# EPICS autosave request: urRobotApp/Db/waypointL_settings.req
$(P)WaypointL:$(N).VAL
$(P)WaypointL:$(N):X.VAL
$(P)WaypointL:$(N):Y.VAL
$(P)WaypointL:$(N):Z.VAL
$(P)WaypointL:$(N):Rx.VAL
$(P)WaypointL:$(N):Ry.VAL
$(P)WaypointL:$(N):Rz.VAL
$(P)WaypointL:$(N):Speed.VAL
$(P)WaypointL:$(N):Acceleration.VAL
$(P)WaypointL:$(N):Blend.VAL
$(P)WaypointL:$(N):Enabled
$(P)WaypointL:$(N):ActionOpt
